// TIA Portal project "newbie" (V15)

(* hardware
DEVICE "S7-1200 station_1"  S7-1200 Station
   slot 0: "Rack_0"  S7-1200 Rack  Rack  V1.0
   slot 1: "PLC_1"  CPU 1214C DC/DC/DC  6ES7 214-1AG40-0XB0  V4.2
DEVICE "HMI_1"  TP900 Comfort
   slot 0: "HMI_1"  TP900 Comfort  6AV2 124-0JC01-0AX0  15.0.0.0
   slot 1: "HMI_RT_1"  TP900 Comfort  6AV2 124-0JC01-0AX0  15.0.0.0
   slot 5: "HMI_1.IE_CP_1"  PROFINET Interface  15.0.0.0
      slot 1: "PROFINET Interface_1"  PROFINET Interface
         slot 1: "Port_1"  Port
         slot 2: "Port_2"  Port
   slot 7: "HMI_1.MPI/DP_CP_1"  MPI/DP Interface  15.0.0.0
*)

// ===== PLC "PLC_1"  CPU 1214C DC/DC/DC =====

VAR_GLOBAL   // PLC tag table "Default tag table"
   "Stop" AT %M0.0 : Bool;
   "Start" AT %M0.1 : Bool;
   "motor1" AT %Q0.0 : Bool;
   "motor2" AT %Q0.1 : Bool;
   "resetauto" AT %M0.2 : Bool;
   "gate" AT %Q0.3 : Bool;
   "sensor" AT %M0.4 : Bool;
   "Tag_1" AT %M0.7 : Bool;
   "active" AT %M1.0 : Bool;
   "Tag_2" AT %MD50 : DInt;
   "tgdem" AT %M0.3 : Bool;
   "resetatc" AT %M0.5 : Bool;
   "Tag_3" AT %M30.0 : Bool;
END_VAR

DATA_BLOCK "Data_block_1"   // DB3
{ S7_Optimized_Access := 'TRUE' }
VERSION : 0.1
   VAR
      ET : DInt;
   END_VAR
BEGIN
END_DATA_BLOCK

// folder: System blocks/Program resources

DATA_BLOCK "IEC_Counter_0_DB"   // DB1
{ S7_Optimized_Access := 'TRUE' }
AUTHOR : Simatic
FAMILY : IEC
NAME : CNTR
VERSION : 1.0
// stored: InstanceOfName IEC_COUNTER
"IEC_COUNTER"
BEGIN
END_DATA_BLOCK

DATA_BLOCK "IEC_Timer_0_DB"   // DB2
{ S7_Optimized_Access := 'TRUE' }
AUTHOR : Simatic
FAMILY : IEC
NAME : IEC_TMR
VERSION : 1.0
// stored: InstanceOfName IEC_TIMER
"IEC_TIMER"
BEGIN
END_DATA_BLOCK

// folder: (top level)

FUNCTION "Block_1" : Void   // FC1, LAD
{ S7_Optimized_Access := 'TRUE' }
VERSION : 0.1
BEGIN
END_FUNCTION

ORGANIZATION_BLOCK "Main"   // OB1, LAD, ProgramCycle
TITLE = "Main Program Sweep (Cycle)"
{ S7_Optimized_Access := 'TRUE' }
VERSION : 0.1
   VAR_INPUT
      Initial_Call : Bool;   // Initial call of this OB
      Remanence : Bool;   // =True, if remanent data are available
   END_VAR
   VAR_TEMP   // added for the SCL form of the ladder/FBD networks
      _w1 : Bool;
      _w2 : Bool;
   END_VAR
BEGIN

REGION Network 1
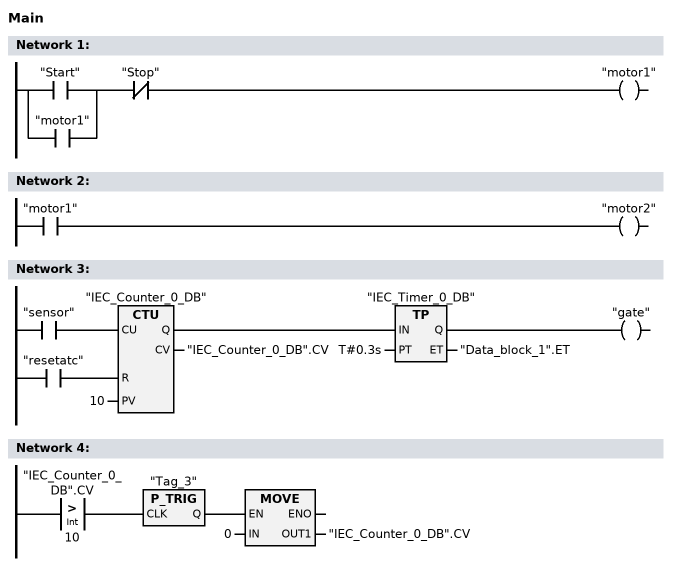
   RUNG wire#powerrail
      Contact( "Start" )
      wire#w1
      I_Contact( "Stop" )
      Coil( "motor1" )
   END_RUNG
   RUNG wire#powerrail
      Contact( "motor1" )
   END_RUNG wire#w1
   // the same network as SCL:
   "motor1" := ("Start" OR "motor1") AND NOT "Stop";
END_REGION

REGION Network 2
   RUNG wire#powerrail
      Contact( "motor1" )
      Coil( "motor2" )
   END_RUNG
   // the same network as SCL:
   "motor2" := "motor1";
END_REGION

REGION Network 3
   "IEC_Counter_0_DB".CTU(CU := "sensor", R := "resetatc", PV := 10, CV => "IEC_Counter_0_DB".CV);
   "IEC_Timer_0_DB".TP(IN := "IEC_Counter_0_DB".Q, PT := T#0.3s, ET => "Data_block_1".ET);
   "gate" := "IEC_Timer_0_DB".Q;
END_REGION

REGION Network 4
   RUNG wire#powerrail
      { S7_Templates := "SrcType := Int" } GT_Contact(in1 := "IEC_Counter_0_DB".CV, in2 := 10)
      P_Trig( "Tag_3" )
      Move(in := 0, out1 => "IEC_Counter_0_DB".CV)
   END_RUNG
   // the same network as SCL:
   #_w1 := "IEC_Counter_0_DB".CV > 10;
   #_w2 := #_w1 AND NOT "Tag_3";   // rising edge
   "Tag_3" := #_w1;
   IF #_w2 THEN "IEC_Counter_0_DB".CV := 0; END_IF;
END_REGION
END_ORGANIZATION_BLOCK

(* ===== HMI "HMI_RT_1" =====
system functions are stored by id; their names below are inferred from use

HMI tags "Default tag table"
   "Start" : Bool = PLC Start AT %M0.1
   "Stop" : Bool = PLC Stop AT %M0.0

screen "Root screen" 800x480, template "Template_1"
   TextField "HmiScreenItemData" at 80,226 size 640x22; Text 'Welcome to HMI_1 (TP900 Comfort)!'
   Button "Button_1" at 14,16 size 96x32; TextOff 'Start'
      on Press: SetBit("Start")
      on Release: ResetBit("Start")
   Button "Button_2" at 14,64 size 96x32; TextOff 'Stop'
      on Press: SetBit("Stop")
      on Release: ResetBit("Stop")
   SymbolLibrary "Symbol library_1" at 147,189 size 120x120

screen "Screen_1" 800x480
   Switch "Switch_1" at 11,17 size 120x57; CaptionText 'Switch'; TextOff 'OFF'; TextOn 'ON'
      on SwitchOn: SetBit("Start")
      on SwitchOff: SetBit("Stop")
   SymbolLibrary "Symbol library_1" at 402,319 size 38x113
   SymbolLibrary "Symbol library_2" at 117,111 size 620x119
   SymbolLibrary "Symbol library_3" at 101,211 size 58x60
   SymbolLibrary "Symbol library_4" at 482,271 size 120x120
*)